FUNCTION_BLOCK FB_LamparaMemorizada_SFC
// La lampara se enciende al accionar el pulsador de conexion
// La lampara se apaga al accionar el pulsador de desconexion
VAR
    Lampara AT %Q*: BOOL;
    PulsadorConexion AT %I*: BOOL;
    PulsadorDesconexion AT %I*: BOOL;
END_VAR

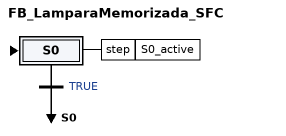
INITIAL_STEP S0:
    S0_active(N);  // step action
END_STEP
TRANSITION FROM S0 TO S0
    := TRUE;
END_TRANSITION

ACTION S0_active:
IF PulsadorDesconexion THEN
    Lampara := FALSE;
ELSIF PulsadorConexion THEN
    Lampara := TRUE;
END_IF
END_ACTION

END_FUNCTION_BLOCK

(* stored: Version 1.1.0.1, ProductVersion 3.1.4024.15
   POU FB_LamparaMemorizada_SFC: Id {7267c7d0-0775-4cd7-b05c-82663a71536c}, SpecialFunc None
   Action S0_active: Id {2bf5d367-24ee-4b2d-946a-fc19475c8227} *)
